TYPE ST_TCPConnection_HMI_Status :
STRUCT
	bCameraReadSocketIsConnected	:BOOL;
	bHlzWriteSocketIsConnected		:BOOL;
	
	aEANRegistry					:ARRAY[0..GVL_Constant.ITEM_ARRAY_SIZE] OF T_MaxString;
END_STRUCT
END_TYPE

(* stored: Version 1.1.0.1, ProductVersion 3.1.4024.12
   DUT ST_TCPConnection_HMI_Status: Id {a398a78d-1809-4dea-8951-d89129f51908} *)
